// TIA Portal V19 export
FUNCTION "ResetPopupBlock" : Void   // FC37, STL
TITLE = Reset start blocking pop up text to intouch PC
{ S7_Optimized_Access := 'TRUE' }
AUTHOR : FLA
FAMILY : UHT
VERSION : 1.0
// FC 36 setup the timer to 5 seconds
// 
// FC 37 reset all text numbers after 5 seconds, and load the value -1 as oneshot 
// 
// M 2.0 uses as 1 hz oneshot
// 
// Programmer Init: 8953-FLA
// 
// Change Log:
// 
// Date        Change                          Updated by
// ------------------------------------------------------
// 19.04.99    1. Edition                      FLA
// stored: AutoNumber false
   VAR_INPUT
      TRIGGER_BIT_1HZ : Bool;   // 1 HZ trigger bit (oneshot)
   END_VAR
BEGIN

NETWORK
TITLE = 
      L     -1;
      L     "PopUpBitToScada".Count_down_to_reset;  // Reset text number count down
      ==I;
      BEC;  // Text numbers already reset

      AN    #TRIGGER_BIT_1HZ;  // 1 hz one shot
      BEC;

      L     1;
      -I;
      T     "PopUpBitToScada".Count_down_to_reset;  // Reset text number count down

      L     0;
      >I;
      BEC;

      L     -1;
      T     "PopUpBitToScada".Count_down_to_reset;  // Do only reset one time

      L     0;
      T     "PopUpBitToScada".Pop_up_text_to_PC1;  // Reset text number to PC 1
      T     "PopUpBitToScada".Pop_up_text_to_PC2;  // Reset text number to PC 2
      T     "PopUpBitToScada".Pop_up_text_to_PC3;  // Reset text number to PC 3
      T     "PopUpBitToScada".Pop_up_text_to_PC4;  // Reset text number to PC 4
      T     "PopUpBitToScada".Pop_up_text_to_PC5;  // Reset text number to PC 5
      T     "PopUpBitToScada".Pop_up_text_to_PC6;  // Reset text number to PC 6
      T     "PopUpBitToScada".Pop_up_text_to_PC7;  // Reset text number to PC 7
      T     "PopUpBitToScada".Pop_up_text_to_PC8;  // Reset text number to PC 8
END_FUNCTION
